{attribute 'qualified_only'}
{attribute 'strict'}
{attribute 'to_string'}
TYPE ST115_Cylinders_e :
(
    GreiferLinks,
    GreiferRechts,
    _max
);
END_TYPE

(* stored: Version 1.1.0.1, ProductVersion 3.1.4024.6
   EnumerationTextList ST115_Cylinders_e: Id {0dac8e02-5f34-492a-a5a1-960ee968f78b} *)
